FUNCTION_BLOCK PUBLIC FB_DevAnalogOutput EXTENDS FB_DevBase 
VAR_INPUT
	fCmdValue		: LREAL := 0 ;
END_VAR
VAR_OUTPUT
	fOutputValue	: LREAL := 0 ;
END_VAR
VAR
	nLimitMin		: INT := -32767 ;
	nLimitMax 		: INT := 32767 ;
	qnHwOut	AT%Q*	: INT := 0 ;
END_VAR

// set device type
IF eDevType = E_Devices.Undefined THEN 
	eDevType := E_Devices.AnalogOut ;
END_IF

// Call base function
SUPER^(refFbFault := refFbFault);


// Call private functions
ExecSetOutput();
ExecSetFeedback();

METHOD INTERNAL ExecSetFeedback : BOOL
VAR_INPUT
END_VAR
// Set feedback 
fOutputValue := INT_TO_LREAL(qnHwOut) ;
END_METHOD

METHOD INTERNAL ExecSetOutput : BOOL
VAR_INPUT
END_VAR
// Set Output to physical device
IF bEnable OR bCmdManual THEN 
	qnHwOut := LREAL_TO_INT(fCmdValue) ; 
	qnHwOut := LIMIT(nLimitMin, qnHwOut, nLimitMax) ; 
ELSE 
	fCmdValue := 0 ; 
END_IF
END_METHOD

END_FUNCTION_BLOCK

(* stored: Version 1.1.0.1, ProductVersion 3.1.4024.5
   POU FB_DevAnalogOutput: Id {c04f47fb-753a-07c6-1304-4d37cf041c4c}, SpecialFunc None
   Folder Private: Id {81264718-d2cd-06cb-14d3-b5473936a556}
   Method ExecSetFeedback: Id {18d9da84-4902-013f-1733-290381c8418e}
   Method ExecSetOutput: Id {72b429d8-82f0-0371-2b55-cc7f874d4b35} *)
